TYPE "PPrf_A0304_0304_Scarico"
VERSION : 0.1
// Block: PPrf_A0304_0304_Scarico
   STRUCT
      Trasporto : PPrf_A0303_Trasporto;
      Navetta : PPrf_A0304_Navetta;
   END_STRUCT;

END_TYPE
